// TIA Portal V16 export
// export: Created 2024-06-24T15:42:27.6675054Z, ExportSetting WithDefaults, DisplayName Totally Integrated Automation Portal, DisplayVersion V16, DisplayName TIA Portal Version Control Interface, DisplayVersion V16, DisplayName TIA Portal Openness, DisplayVersion V16, DisplayName STEP 7 Professional, DisplayVersion V16, DisplayName STEP 7 Safety, DisplayVersion V16, DisplayName WinCC Advanced, DisplayVersion V16
ORGANIZATION_BLOCK "OB_Machine_Ready"   // OB126, LAD, ProgramCycle
TITLE = "Main Program Sweep (Cycle)"
{ S7_Optimized_Access := 'TRUE' }
VERSION : 0.1
// stored: AutoNumber true, IsIECCheckEnabled false, SetENOAutomatically false
   VAR_INPUT
      Initial_Call : Bool;   // Initial call of this OB
      Remanence : Bool;   // =True, if remanent data are available
   END_VAR
BEGIN

REGION Network 1
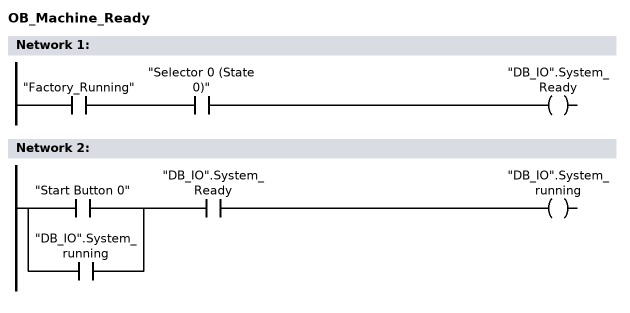
   RUNG wire#powerrail
      Contact( "Factory_Running" )
      Contact( "Selector 0 (State 0)" )
      Coil( "DB_IO".System_Ready )
   END_RUNG
   // the same network as SCL:
   "DB_IO".System_Ready := "Factory_Running" AND "Selector 0 (State 0)";
END_REGION

REGION Network 2
   RUNG wire#powerrail
      Contact( "Start Button 0" )
      wire#w1
      Contact( "DB_IO".System_Ready )
      Coil( "DB_IO".System_running )
   END_RUNG
   RUNG wire#powerrail
      Contact( "DB_IO".System_running )
   END_RUNG wire#w1
   // the same network as SCL:
   "DB_IO".System_running := ("Start Button 0" OR "DB_IO".System_running) AND "DB_IO".System_Ready;
END_REGION
END_ORGANIZATION_BLOCK
